(*
SPDX-FileCopyrightText: © 2026 Oleksandr Tiutyk <trofimich@gmail.com>
SPDX-License-Identifier: MIT
License: https://opensource.org/license/mit
*)

(*!
<summary>Checks whether a filesystem directory exists through cyclic task execution.</summary>
<description>
Stopping closes an unfinished native enumeration before reporting completion. Diagnostic string inputs are
borrowed only during the call; retained diagnostic text is copied into owned storage. A found file is a
successful check with DirectoryExists=FALSE.
</description>
*)

{attribute 'no_explicit_call' := 'do not call this function block directly'}
FUNCTION_BLOCK CheckDirectoryExists EXTENDS TOF_Tasks.Task IMPLEMENTS IFileSystemTask
VAR_STAT
	//! <summary>Static type metadata available before the base task initializes its default name.</summary>
	{attribute 'hide'}
	_ClassName : STRING := __POUNAME();
END_VAR
VAR
	_EnumFindFile : Tc2_Utilities.FB_EnumFindFileEntry;
	//! <summary>Records whether a search command may still own native enumeration resources.</summary>
	_EnumerationStarted : BOOL;
	//! <summary>Prevents repeating the abort command while its completion is pending.</summary>
	_EnumerationAbortIssued : BOOL;
	
	_DirectoryExists : BOOL;
END_VAR

(*!
<summary>Selects the ADS target for the native filesystem operation.</summary>
<description>
Configure before Start and keep unchanged until STOPPED; the setter stores configuration without submitting
I/O.
</description>
*)
{attribute 'monitoring' := 'call'}
PROPERTY AmsNetId : Tc2_System.T_AmsNetID
GET
AmsNetId := _EnumFindFile.sNetId;
END_GET
SET
_EnumFindFile.sNetId := AmsNetId;
END_SET
END_PROPERTY

(*!
<summary>Provides the concrete type name used in diagnostics.</summary>
<description>
Returns borrowed read-only metadata; keep the instance alive and do not modify the referenced string.
Initialized static storage is ready during base Task.FB_init; this getter has no side effects or exceptions.
</description>
*)
{attribute 'monitoring' := 'call'}
PROPERTY ClassName : REFERENCE TO STRING
GET
ClassName REF= _ClassName;
END_GET
END_PROPERTY

(*!
<summary>Reports whether the completed check found a directory.</summary>
<description>
Meaningful after successful task completion. FALSE means no entry or a found file; a failed search must be
distinguished through FinalStopReason. Reset clears this result.
</description>
*)
{attribute 'monitoring' := 'call'}
PROPERTY DirectoryExists : BOOL
GET
DirectoryExists := _DirectoryExists;
END_GET
END_PROPERTY

(*!
<summary>Provides the copied directory path used by the operation and its existence check.</summary>
<description>
Configure before Start and keep unchanged until STOPPED. PathHelper applies its limited lexical filter before
native submission. Assignment does not perform I/O; Reset preserves the path.
</description>
*)
{attribute 'monitoring' := 'call'}
PROPERTY DirectoryPath : Tc2_System.T_MaxString
GET
DirectoryPath := _EnumFindFile.sPathName;
END_GET
SET
_EnumFindFile.sPathName := DirectoryPath;
END_SET
END_PROPERTY

(*!
<summary>Provides the library namespace used in diagnostics.</summary>
<description>Returns borrowed read-only namespace storage; do not modify the referenced string.</description>
*)
{attribute 'monitoring' := 'call'}
PROPERTY NamespaceName : REFERENCE TO STRING
GET
NamespaceName REF= CurrentNamespace.Name;
END_GET
END_PROPERTY

(*!
<summary>Clears the completed search and its per-run cleanup state for reuse.</summary>
<description>Called only after stopping has completed; it does not abandon a pending enumeration command.</description>
*)
METHOD PROTECTED OnReset
_EnumFindFile(bExecute := FALSE);

_EnumerationStarted := FALSE;
_EnumerationAbortIssued := FALSE;
_DirectoryExists := FALSE;
END_METHOD

(*!
<summary>Checks one directory search and reports whether the found entry is a directory.</summary>
<description>
Starts the search once, then advances it until an entry, end-of-enumeration or error is reported. A found file
leaves DirectoryExists=FALSE and completes successfully. Early completion leaves native enumeration cleanup to
OnStopping. Computed diagnostics are held in local buffers for the duration of the receiving call without
dynamic string-builder allocations.
</description>
<param name="processingState">DONE after a completed search; BUSY while the command is pending.</param>
<param name="stopReasonMessage">Not changed; exceptions provide search failure diagnostics.</param>
*)
METHOD PROTECTED OnRunning
VAR_OUTPUT
	processingState : TOF_Tasks.TASK_PROCESSING_STATE;
END_VAR
VAR_IN_OUT
	stopReasonMessage : TOF_Core.ERROR_MESSAGE;
END_VAR
VAR	
	pathErrorMessage : WSTRING(255);
	formattedExceptionMessage : TOF_Core.ERROR_MESSAGE;
END_VAR
IF NOT _EnumFindFile.bExecute THEN 
	IF TOF_Core.Strings.IsNullOrWhiteSpace(stringToCheck := _EnumFindFile.sPathName) THEN
		TOF_Core.Exceptions.ThrowDataMemberNotSpecified(
			sourceNamespaceName := NamespaceName,
			sourceClassName := ClassName,
			sourcePOUName := __POUNAME(),
			sourcePosition := __POSITION(),
			dataMemberName := 'DirectoryPath'
		);		
	END_IF
	
	IF NOT PathHelper.IsValidDirectoryPath(directoryPath := _EnumFindFile.sPathName, errorMessage => pathErrorMessage) THEN
		FileSystemExceptions.ThrowInvalidPath(
			sourceNamespaceName := NamespaceName,
			sourceClassName := ClassName,
			sourcePOUName := __POUNAME(),
			sourcePosition := __POSITION(),
			path := _EnumFindFile.sPathName,
			errorMessage := pathErrorMessage
		);
	END_IF
	
	_EnumFindFile.eCmd := Tc2_Utilities.E_EnumCmdType.eEnumCmd_First;
END_IF

_EnumerationStarted := TRUE;
_EnumFindFile(bExecute := TRUE);

IF _EnumFindFile.bError THEN
	TOF_Core.WideStrings.Append255(
		formattedExceptionMessage,
		"Error while checking directory '",
		TO_WSTRING(_EnumFindFile.sPathName),
		"'");

	FileSystemExceptions.ThrowFileSystem(
		sourceNamespaceName := NamespaceName,
		sourceClassName := ClassName,
		sourcePOUName := __POUNAME(),
		sourcePosition := __POSITION(),
		message := formattedExceptionMessage,
		errorCode := _EnumFindFile.nErrId
	);
ELSIF NOT _EnumFindFile.bBusy THEN	
	IF NOT _EnumFindFile.bEOE THEN
		_DirectoryExists := _EnumFindFile.stFindFile.fileAttributes.bDirectory;		
	END_IF

	processingState := TOF_Tasks.TASK_PROCESSING_STATE.DONE;
END_IF
END_METHOD

(*!
<summary>Advances directory stop actions before reporting termination.</summary>
<description>
Used for every stop reason. Drains a pending search before deciding whether its native enumeration must be
aborted. An unfinished search receives one abort command with a rising bExecute edge; readiness waits for that
command to complete. End-of-enumeration and search errors need no explicit abort. No new search starts. An
abort error is logged once with its native code and path, without retrying abort or replacing the task stop
reason. Readiness means this cleanup attempt ended, not that server resources were proven released. The log
attempt is made after clearing pending enumeration state; logger failure does not restart cleanup.
</description>
<param name="readyToRelease">TRUE when the directory FBs have finished their pending requests.</param>
*)
METHOD PROTECTED OnStopping
VAR_OUTPUT
	readyToRelease : BOOL;
END_VAR
VAR
	enumerationAbortMessage : WSTRING(255);
END_VAR
IF _EnumerationStarted THEN
	_EnumFindFile(bExecute := FALSE);

	IF NOT _EnumFindFile.bBusy THEN
		IF _EnumFindFile.bEOE OR_ELSE _EnumFindFile.bError THEN
			_EnumerationStarted := FALSE;

			(* End this attempt before reporting its error so logging cannot cause repeated aborts. *)
			IF _EnumerationAbortIssued AND_THEN _EnumFindFile.bError THEN
				enumerationAbortMessage := TOF_Core.WideStrings.Concat255(
					"Directory enumeration abort failed (native error code ",
					TO_WSTRING(_EnumFindFile.nErrId),
					"): ",
					TO_WSTRING(_EnumFindFile.sPathName)
				);
				TOF_Core.LogManager.TryLogMessage(
					message := enumerationAbortMessage,
					category := TOF_Core.LOG_CATEGORY.ERROR,
					topic1 := TO_WSTRING(__POUNAME())
				);
			END_IF
		ELSIF NOT _EnumerationAbortIssued THEN
			_EnumFindFile(bExecute := TRUE, eCmd := Tc2_Utilities.E_EnumCmdType.eEnumCmd_Abort);
			_EnumerationAbortIssued := TRUE;
		ELSE
			_EnumerationStarted := FALSE;
		END_IF
	END_IF
END_IF

readyToRelease := NOT _EnumerationStarted;
END_METHOD

(*!
<summary>Selects the native path context for the filesystem request.</summary>
<description>
Configure before Start and keep unchanged until STOPPED. It is passed to the native operation, not used as a
path-validity result. Reset preserves it. Target support includes the ePath enumeration input in
Tc2_Utilities 3.10.9.
</description>
*)
{attribute 'monitoring' := 'call'}
PROPERTY PathType : Tc2_System.E_OpenPath
GET
PathType := _EnumFindFile.ePath;
END_GET
SET
_EnumFindFile.ePath := PathType;
END_SET
END_PROPERTY

(*!
<summary>Reports the size of this concrete instance in bytes.</summary>
*)
{attribute 'monitoring' := 'call'}
PROPERTY SelfSize : ULINT
GET
SelfSize := XSIZEOF(THIS^);
END_GET
END_PROPERTY

(*!
<summary>Configures the timeout passed to native operation requests.</summary>
<description>
Set before Start and keep unchanged until STOPPED. Reset preserves this value. It is not an overall task
deadline or a guarantee of resource release after a timeout.
</description>
*)
{attribute 'monitoring' := 'call'}
PROPERTY Timeout : TIME
GET
Timeout := _EnumFindFile.tTimeout;
END_GET
SET
_EnumFindFile.tTimeout := Timeout;
END_SET
END_PROPERTY

END_FUNCTION_BLOCK

(* stored: Version 1.1.0.1
   POU CheckDirectoryExists: Id {e725df2c-ff5d-4b1a-879a-c0e9431a08b3}, SpecialFunc None
   Folder Inputs: Id {540d797c-4279-445e-aff3-e32f9993a17f}
   Folder Members to override: Id {f7ddb29a-7136-4b3e-8b27-52a98a0c5305}
   Folder Outputs: Id {0cec064e-0e57-41f5-ae10-54ef9890bc2e}
   Property AmsNetId: Id {2728b040-bcd8-4512-9b72-dde642a14465}
   Get Get: Id {292fd92d-b98c-4b24-8439-f7025d4ee4ac}
   Set Set: Id {192383b9-1553-4a0e-90e9-1629accbcba8}
   Property ClassName: Id {58a4a779-e96f-4151-9f98-191872bf5430}
   Get Get: Id {f2b48812-6ff9-4d66-a895-e968f44a2c9a}
   Property DirectoryExists: Id {93f1f338-f94f-430f-b1d1-ddbe863c8b22}
   Get Get: Id {adc8b4d3-4be0-4245-95f4-c54d6d0787ca}
   Property DirectoryPath: Id {9371e100-c77a-4bcb-a00b-81c8f661f34e}
   Get Get: Id {09f16cb5-8893-4e5c-b803-d96e500c8198}
   Set Set: Id {35bc8e6d-793a-4dce-afdb-edb7f38eb71e}
   Property NamespaceName: Id {9e94954c-e994-471e-a045-591284438b65}
   Get Get: Id {b6141f2c-59cb-43ba-9c85-87eeb2c85167}
   Method OnReset: Id {fe840260-57c7-49f3-acb3-979b08331a03}
   Method OnRunning: Id {a2b5ac80-a25f-47e6-8333-9adc249a4985}
   Method OnStopping: Id {3f5e6d21-6c7f-4e76-a89e-10f3fb296d85}
   Property PathType: Id {9772faee-bff2-418a-bc6a-dee866cc52c7}
   Get Get: Id {06f502d4-7292-4eba-805f-ca3c5508de2b}
   Set Set: Id {71ca7076-0db4-4dcb-aa15-e105c679e3b8}
   Property SelfSize: Id {6747bc52-107d-4a38-b726-e67926a684e4}
   Get Get: Id {f6bf50fb-a7d1-4bbf-8d89-c812dbd5b80d}
   Property Timeout: Id {f4c81150-54ac-4b5e-8bd7-df7a33619591}
   Get Get: Id {c11a20a4-9bf7-49d2-8382-5ba592399554}
   Set Set: Id {14d878ec-05ac-405f-881a-8d4f4ccde574} *)
